{attribute 'pack_mode' := '1'} 
// ------------------------------------------------------------------------- 
//  SRCI Robot Library                                                
// ------------------------------------------------------------------------- 
//                                                                           
//  Object:      ReadAnalogInputOutCmd                                       
//  Author:      Thorsten Brach                                                
//  Date:        2024-08-09
//
//  Description:                                              
//   
//                                                                           
//  Copyright: 
//    (C) 2024 Thorsten Brach. All rights reserved                                                                                                                                            
//             Licensed under the MIT License.
//                                                                           
//  Disclaimer:                                                                           
//    This project is provided without any guarantee and can be used for   
//    private and commercial purposes. Any use is at the user’s 
//    own risk and responsibility.
//
// -------------------------------------------------------------------------
TYPE ReadAnalogInputOutCmd :
STRUCT
  /// Relates to ListenerID >0 
  /// Number of successful trigger -based command invocations
  /// For more information refer to chapter 5.5.12.4.
  InvocationCounter  : USINT;
  /// Unique system-generated ID of the "Action" when the function is triggered.
  /// • >0: The "Action" is started by the trigger funcrion with identical FollowID.
  /// • <0: The "Action" is stopped by the trigger function with identical FollowID.
  /// For more information see chapter 5.5.12.4 EmitterID, ListenerID, FollowID and OriginID
  OriginID           : INT;
  /// Returned values of digital inputs
  /// Returned values of digital inputs
  /// Unit of returned Value
  Unit               : UnitType;
  /// Returned value of analog input
  Value              : REAL;
END_STRUCT
END_TYPE

{attribute 'pack_mode' := '1'} 
// ------------------------------------------------------------------------- 
//  SRCI Robot Library                                                
// ------------------------------------------------------------------------- 
//                                                                           
//  Object:      ReadAnalogInputParCmd                                       
//  Author:      Thorsten Brach                                                
//  Date:        2024-08-09
//
//  Description:                                              
//   
//                                                                           
//  Copyright: 
//    (C) 2024 Thorsten Brach. All rights reserved                                                                                                                                            
//             Licensed under the MIT License.
//                                                                           
//  Disclaimer:                                                                           
//    This project is provided without any guarantee and can be used for   
//    private and commercial purposes. Any use is at the user’s 
//    own risk and responsibility.
//
// -------------------------------------------------------------------------
TYPE ReadAnalogInputParCmd :
STRUCT
  /// Number of the analog input 1..32
  Index              : USINT; 
  /// ID of associated trigger function:
  /// •  0: No Trigger (default)  No trigger related behavior
  /// • >0: Trigger - Start executing when the trigger function with the identical EmitterID is triggered.
  /// Always positive.
  /// For more information, see chapter 5.5.12 Triggers
  ListenerID         : SINT;
END_STRUCT
END_TYPE

{attribute 'pack_mode' := '1'} 
// ------------------------------------------------------------------------- 
//  SRCI Robot Library                                                
// ------------------------------------------------------------------------- 
//                                                                           
//  Object:      ReadAnalogInputRecvData                                       
//  Author:      Thorsten Brach                                                
//  Date:        2024-08-09
//
//  Description:                                              
//   
//                                                                           
//  Copyright: 
//    (C) 2024 Thorsten Brach. All rights reserved                                                                                                                                            
//             Licensed under the MIT License.
//                                                                           
//  Disclaimer:                                                                           
//    This project is provided without any guarantee and can be used for   
//    private and commercial purposes. Any use is at the user’s 
//    own risk and responsibility.
//
// -------------------------------------------------------------------------
TYPE ReadAnalogInputRecvData EXTENDS RspHeader :
STRUCT
  /// Relates to ListenerID >0
  /// Number of successful trigger-based command invocations - For more information refer TO chapter 5.5.12.4
  InvocationCounter : USINT;  
  /// Reserve
  Reserve           : SINT;
  /// Unique system-generated ID of the "Action" when the function is triggered.
  /// • >0: The "Action" is started by the trigger funcrion with identical FollowID.
  /// • <0: The "Action" is stopped by the trigger function with identical FollowID.
  /// For more information see chapter 5.5.12.4 EmitterID, ListenerID, FollowID and OriginID
  OriginID          : INT;
  /// Returned values of digital inputs
  /// Returned values of digital inputs
  /// Unit of returned Value
  Unit               : USINT;
  /// Returned value of analog input
  Value              : REAL;  
END_STRUCT
END_TYPE

{attribute 'pack_mode' := '1'}
// ------------------------------------------------------------------------- 
//  SRCI Robot Library                                                
// ------------------------------------------------------------------------- 
//                                                                           
//  Object:      ReadAnalogInputSendData                                       
//  Author:      Thorsten Brach                                                
//  Date:        2024-08-09
//
//  Description:                                              
//   
//                                                                           
//  Copyright: 
//    (C) 2024 Thorsten Brach. All rights reserved                                                                                                                                            
//             Licensed under the MIT License.
//                                                                           
//  Disclaimer:                                                                           
//    This project is provided without any guarantee and can be used for   
//    private and commercial purposes. Any use is at the user’s 
//    own risk and responsibility.
//
// -------------------------------------------------------------------------
TYPE ReadAnalogInputSendData EXTENDS CmdHeader: 
STRUCT
  /// ID of Action that will be executed when this command is active
  /// • >0: Start Action - Start executing the Action function with the identical ListenerID.
  /// • <0: Stop Action  -  Stop executing the Action function with the identical ListenerID.
  /// • 0: No trigger (default)-  If no EmitterID is defined, the function will not trigger any Action during its execution
  /// For more information see section Triggers of this chapter or chapter 5.5.12.4.
  EmitterID          : ARRAY [0..3] OF SINT;
  /// ID of associated trigger function:
  /// •  0: No Trigger (default)  No trigger related behavior
  /// • >0: Trigger - Start executing when the trigger function with the identical EmitterID is triggered.
  /// Always positive.
  /// For more information, see chapter 5.5.12 Triggers
  ListenerID         : SINT;
  /// Reserve
  Reserve            : BYTE;
  /// Number of the analog input 1..32
  Index              : USINT; 
END_STRUCT
END_TYPE

{attribute 'pack_mode' := '1'} 
// ------------------------------------------------------------------------- 
//  SRCI Robot Library                                                
// ------------------------------------------------------------------------- 
//                                                                           
//  Object:      ReadDigitalInputsOutCmd                                       
//  Author:      Thorsten Brach                                                
//  Date:        2024-08-09
//
//  Description:                                              
//   
//                                                                           
//  Copyright: 
//    (C) 2024 Thorsten Brach. All rights reserved                                                                                                                                            
//             Licensed under the MIT License.
//                                                                           
//  Disclaimer:                                                                           
//    This project is provided without any guarantee and can be used for   
//    private and commercial purposes. Any use is at the user’s 
//    own risk and responsibility.
//
// -------------------------------------------------------------------------
TYPE ReadDHParameterOutCmd :
STRUCT
  /// Denavit–Hartenberg parameter
  DHParameter : DHParameter;
END_STRUCT
END_TYPE

{attribute 'pack_mode' := '1'} 
// ------------------------------------------------------------------------- 
//  SRCI Robot Library                                                
// ------------------------------------------------------------------------- 
//                                                                           
//  Object:      ReadDigitalInputsParCmd                                       
//  Author:      Thorsten Brach                                                
//  Date:        2024-08-09
//
//  Description:                                              
//   
//                                                                           
//  Copyright: 
//    (C) 2024 Thorsten Brach. All rights reserved                                                                                                                                            
//             Licensed under the MIT License.
//                                                                           
//  Disclaimer:                                                                           
//    This project is provided without any guarantee and can be used for   
//    private and commercial purposes. Any use is at the user’s 
//    own risk and responsibility.
//
// -------------------------------------------------------------------------
TYPE ReadDHParameterParCmd :
STRUCT
  /// Determines if returned DH parameters use modified convention or classic convention.
  /// • 0: Classic convention (default)
  /// • 1: Modified convention
  ModifiedConvention : BOOL;  
END_STRUCT
END_TYPE

{attribute 'pack_mode' := '1'} 
// ------------------------------------------------------------------------- 
//  SRCI Robot Library                                                
// ------------------------------------------------------------------------- 
//                                                                           
//  Object:      ReadDigitalInputsRecvData                                       
//  Author:      Thorsten Brach                                                
//  Date:        2024-08-09
//
//  Description:                                              
//   
//                                                                           
//  Copyright: 
//    (C) 2024 Thorsten Brach. All rights reserved                                                                                                                                            
//             Licensed under the MIT License.
//                                                                           
//  Disclaimer:                                                                           
//    This project is provided without any guarantee and can be used for   
//    private and commercial purposes. Any use is at the user’s 
//    own risk and responsibility.
//
// -------------------------------------------------------------------------
TYPE ReadDHParameterRecvData EXTENDS RspHeader :
STRUCT
  /// Denavit–Hartenberg parameter
  DHParameter : DHParameter;  
END_STRUCT
END_TYPE

{attribute 'pack_mode' := '1'}
// ------------------------------------------------------------------------- 
//  SRCI Robot Library                                                
// ------------------------------------------------------------------------- 
//                                                                           
//  Object:      ReadDigitalInputsSendData                                       
//  Author:      Thorsten Brach                                                
//  Date:        2024-08-09
//
//  Description:                                              
//   
//                                                                           
//  Copyright: 
//    (C) 2024 Thorsten Brach. All rights reserved                                                                                                                                            
//             Licensed under the MIT License.
//                                                                           
//  Disclaimer:                                                                           
//    This project is provided without any guarantee and can be used for   
//    private and commercial purposes. Any use is at the user’s 
//    own risk and responsibility.
//
// -------------------------------------------------------------------------
TYPE ReadDHParameterSendData EXTENDS CmdHeader: 
STRUCT
  /// Determines if returned DH parameters use modified convention or classic convention.
  /// • 0: Classic convention (default)
  /// • 1: Modified convention
  ModifiedConvention : BOOL;  
END_STRUCT
END_TYPE

{attribute 'pack_mode' := '1'} 
// ------------------------------------------------------------------------- 
//  SRCI Robot Library                                                
// ------------------------------------------------------------------------- 
//                                                                           
//  Object:      ReadDigitalInputsOutCmd                                       
//  Author:      Thorsten Brach                                                
//  Date:        2024-08-09
//
//  Description:                                              
//   
//                                                                           
//  Copyright: 
//    (C) 2024 Thorsten Brach. All rights reserved                                                                                                                                            
//             Licensed under the MIT License.
//                                                                           
//  Disclaimer:                                                                           
//    This project is provided without any guarantee and can be used for   
//    private and commercial purposes. Any use is at the user’s 
//    own risk and responsibility.
//
// -------------------------------------------------------------------------
TYPE ReadDigitalInputsOutCmd :
STRUCT
  /// Relates to ListenerID >0 
  /// Number of successful trigger -based command invocations
  /// For more information refer to chapter 5.5.12.4.
  InvocationCounter  : USINT;
  /// Unique system-generated ID of the "Action" when the function is triggered.
  /// • >0: The "Action" is started by the trigger funcrion with identical FollowID.
  /// • <0: The "Action" is stopped by the trigger function with identical FollowID.
  /// For more information see chapter 5.5.12.4 EmitterID, ListenerID, FollowID and OriginID
  OriginID           : INT;
  /// Returned values of digital inputs
  Values             : ARRAY[0..4] OF BYTE;
  /// Unique system-generated ID of the "Action" when the function is triggered.
  /// • >0: The "Action" is started by the trigger function with identical FollowID.
  /// • <0: The "Action" is stopped by the trigger function with identical FollowID.
  /// For more information see chapter 5.5.12.4.
END_STRUCT
END_TYPE

{attribute 'pack_mode' := '1'} 
// ------------------------------------------------------------------------- 
//  SRCI Robot Library                                                
// ------------------------------------------------------------------------- 
//                                                                           
//  Object:      ReadDigitalInputsParCmd                                       
//  Author:      Thorsten Brach                                                
//  Date:        2024-08-09
//
//  Description:                                              
//   
//                                                                           
//  Copyright: 
//    (C) 2024 Thorsten Brach. All rights reserved                                                                                                                                            
//             Licensed under the MIT License.
//                                                                           
//  Disclaimer:                                                                           
//    This project is provided without any guarantee and can be used for   
//    private and commercial purposes. Any use is at the user’s 
//    own risk and responsibility.
//
// -------------------------------------------------------------------------
TYPE ReadDigitalInputsParCmd :
STRUCT
  /// Specifies the desired byte addresses that shall be read
  Index              : ARRAY[0..4] OF USINT; 
  /// ID of associated trigger function:
  /// •  0: No Trigger (default)  No trigger related behavior
  /// • >0: Trigger - Start executing when the trigger function with the identical EmitterID is triggered.
  /// Always positive.
  /// For more information, see chapter 5.5.12 Triggers
  ListenerID         : SINT;
END_STRUCT
END_TYPE

{attribute 'pack_mode' := '1'} 
// ------------------------------------------------------------------------- 
//  SRCI Robot Library                                                
// ------------------------------------------------------------------------- 
//                                                                           
//  Object:      ReadDigitalInputsRecvData                                       
//  Author:      Thorsten Brach                                                
//  Date:        2024-08-09
//
//  Description:                                              
//   
//                                                                           
//  Copyright: 
//    (C) 2024 Thorsten Brach. All rights reserved                                                                                                                                            
//             Licensed under the MIT License.
//                                                                           
//  Disclaimer:                                                                           
//    This project is provided without any guarantee and can be used for   
//    private and commercial purposes. Any use is at the user’s 
//    own risk and responsibility.
//
// -------------------------------------------------------------------------
TYPE ReadDigitalInputsRecvData EXTENDS RspHeader :
STRUCT
  /// Relates to ListenerID >0
  /// Number of successful trigger-based command invocations - For more information refer TO chapter 5.5.12.4
  InvocationCounter : USINT;  
  /// Reserve
  Reserve           : SINT;
  /// Unique system-generated ID of the "Action" when the function is triggered.
  /// • >0: The "Action" is started by the trigger funcrion with identical FollowID.
  /// • <0: The "Action" is stopped by the trigger function with identical FollowID.
  /// For more information see chapter 5.5.12.4 EmitterID, ListenerID, FollowID and OriginID
  OriginID          : INT;
  /// Returned values of digital inputs
  Values             : ARRAY[0..4] OF BYTE;
  
END_STRUCT
END_TYPE

{attribute 'pack_mode' := '1'}
// ------------------------------------------------------------------------- 
//  SRCI Robot Library                                                
// ------------------------------------------------------------------------- 
//                                                                           
//  Object:      ReadDigitalInputsSendData                                       
//  Author:      Thorsten Brach                                                
//  Date:        2024-08-09
//
//  Description:                                              
//   
//                                                                           
//  Copyright: 
//    (C) 2024 Thorsten Brach. All rights reserved                                                                                                                                            
//             Licensed under the MIT License.
//                                                                           
//  Disclaimer:                                                                           
//    This project is provided without any guarantee and can be used for   
//    private and commercial purposes. Any use is at the user’s 
//    own risk and responsibility.
//
// -------------------------------------------------------------------------
TYPE ReadDigitalInputsSendData EXTENDS CmdHeader: 
STRUCT
  /// ID of Action that will be executed when this command is active
  /// • >0: Start Action - Start executing the Action function with the identical ListenerID.
  /// • <0: Stop Action  -  Stop executing the Action function with the identical ListenerID.
  /// • 0: No trigger (default)-  If no EmitterID is defined, the function will not trigger any Action during its execution
  /// For more information see section Triggers of this chapter or chapter 5.5.12.4.
  EmitterID          : ARRAY [0..3] OF SINT;
  /// ID of associated trigger function:
  /// •  0: No Trigger (default)  No trigger related behavior
  /// • >0: Trigger - Start executing when the trigger function with the identical EmitterID is triggered.
  /// Always positive.
  /// For more information, see chapter 5.5.12 Triggers
  ListenerID         : SINT;
  /// Reserve
  Reserve            : BYTE;
  /// Specifies the desired byte addresses that shall be read
  Index              : ARRAY[0..4] OF USINT;
END_STRUCT
END_TYPE

{attribute 'pack_mode' := '1'} 
// ------------------------------------------------------------------------- 
//  SRCI Robot Library                                                
// ------------------------------------------------------------------------- 
//                                                                           
//  Object:      ReadDigitalOutputsOutCmd                                       
//  Author:      Thorsten Brach                                                
//  Date:        2024-08-09
//
//  Description:                                              
//   
//                                                                           
//  Copyright: 
//    (C) 2024 Thorsten Brach. All rights reserved                                                                                                                                            
//             Licensed under the MIT License.
//                                                                           
//  Disclaimer:                                                                           
//    This project is provided without any guarantee and can be used for   
//    private and commercial purposes. Any use is at the user’s 
//    own risk and responsibility.
//
// -------------------------------------------------------------------------
TYPE ReadDigitalOutputsOutCmd :
STRUCT
  /// Relates to ListenerID >0 
  /// Number of successful trigger -based command invocations
  /// For more information refer to chapter 5.5.12.4.
  InvocationCounter  : USINT;
  /// Unique system-generated ID of the "Action" when the function is triggered.
  /// • >0: The "Action" is started by the trigger funcrion with identical FollowID.
  /// • <0: The "Action" is stopped by the trigger function with identical FollowID.
  /// For more information see chapter 5.5.12.4 EmitterID, ListenerID, FollowID and OriginID
  OriginID           : INT;
  /// Returned values of digital inputs
  Values             : ARRAY[0..4] OF BYTE;
END_STRUCT
END_TYPE

{attribute 'pack_mode' := '1'} 
// ------------------------------------------------------------------------- 
//  SRCI Robot Library                                                
// ------------------------------------------------------------------------- 
//                                                                           
//  Object:      ReadDigitalOutputsParCmd                                       
//  Author:      Thorsten Brach                                                
//  Date:        2024-08-09
//
//  Description:                                              
//   
//                                                                           
//  Copyright: 
//    (C) 2024 Thorsten Brach. All rights reserved                                                                                                                                            
//             Licensed under the MIT License.
//                                                                           
//  Disclaimer:                                                                           
//    This project is provided without any guarantee and can be used for   
//    private and commercial purposes. Any use is at the user’s 
//    own risk and responsibility.
//
// -------------------------------------------------------------------------
TYPE ReadDigitalOutputsParCmd :
STRUCT
  /// Specifies the desired byte addresses that shall be read
  Index              : ARRAY[0..4] OF USINT; 
  /// ID of associated trigger function:
  /// •  0: No Trigger (default)  No trigger related behavior
  /// • >0: Trigger - Start executing when the trigger function with the identical EmitterID is triggered.
  /// Always positive.
  /// For more information, see chapter 5.5.12 Triggers
  ListenerID         : SINT;
END_STRUCT
END_TYPE

{attribute 'pack_mode' := '1'} 
// ------------------------------------------------------------------------- 
//  SRCI Robot Library                                                
// ------------------------------------------------------------------------- 
//                                                                           
//  Object:      ReadDigitalOutputsRecvData                                       
//  Author:      Thorsten Brach                                                
//  Date:        2024-08-09
//
//  Description:                                              
//   
//                                                                           
//  Copyright: 
//    (C) 2024 Thorsten Brach. All rights reserved                                                                                                                                            
//             Licensed under the MIT License.
//                                                                           
//  Disclaimer:                                                                           
//    This project is provided without any guarantee and can be used for   
//    private and commercial purposes. Any use is at the user’s 
//    own risk and responsibility.
//
// -------------------------------------------------------------------------
TYPE ReadDigitalOutputsRecvData EXTENDS RspHeader :
STRUCT
  /// Relates to ListenerID >0
  /// Number of successful trigger-based command invocations - For more information refer TO chapter 5.5.12.4
  InvocationCounter : USINT;  
  /// Reserve
  Reserve           : SINT;
  /// Unique system-generated ID of the "Action" when the function is triggered.
  /// • >0: The "Action" is started by the trigger funcrion with identical FollowID.
  /// • <0: The "Action" is stopped by the trigger function with identical FollowID.
  /// For more information see chapter 5.5.12.4 EmitterID, ListenerID, FollowID and OriginID
  OriginID          : INT;
  /// Returned values of digital inputs
  Values             : ARRAY[0..4] OF BYTE;
END_STRUCT
END_TYPE

{attribute 'pack_mode' := '1'}
// ------------------------------------------------------------------------- 
//  SRCI Robot Library                                                
// ------------------------------------------------------------------------- 
//                                                                           
//  Object:      ReadDigitalOutputsSendData                                       
//  Author:      Thorsten Brach                                                
//  Date:        2024-08-09
//
//  Description:                                              
//   
//                                                                           
//  Copyright: 
//    (C) 2024 Thorsten Brach. All rights reserved                                                                                                                                            
//             Licensed under the MIT License.
//                                                                           
//  Disclaimer:                                                                           
//    This project is provided without any guarantee and can be used for   
//    private and commercial purposes. Any use is at the user’s 
//    own risk and responsibility.
//
// -------------------------------------------------------------------------
TYPE ReadDigitalOutputsSendData EXTENDS CmdHeader: 
STRUCT
  /// ID of Action that will be executed when this command is active
  /// • >0: Start Action - Start executing the Action function with the identical ListenerID.
  /// • <0: Stop Action  -  Stop executing the Action function with the identical ListenerID.
  /// • 0: No trigger (default)-  If no EmitterID is defined, the function will not trigger any Action during its execution
  /// For more information see section Triggers of this chapter or chapter 5.5.12.4.
  EmitterID          : ARRAY [0..3] OF SINT;
  /// ID of associated trigger function:
  /// •  0: No Trigger (default)  No trigger related behavior
  /// • >0: Trigger - Start executing when the trigger function with the identical EmitterID is triggered.
  /// Always positive.
  /// For more information, see chapter 5.5.12 Triggers
  ListenerID         : SINT;
  /// Reserve
  Reserve            : BYTE;
  /// Specifies the desired byte addresses that shall be read
  Index              : ARRAY[0..4] OF USINT; 
END_STRUCT
END_TYPE

{attribute 'pack_mode' := '1'} 
// ------------------------------------------------------------------------- 
//  SRCI Robot Library                                                
// ------------------------------------------------------------------------- 
//                                                                           
//  Object:      ReadDigitalOutputsOutCmd                                       
//  Author:      Thorsten Brach                                                
//  Date:        2024-08-09
//
//  Description:                                              
//   
//                                                                           
//  Copyright: 
//    (C) 2024 Thorsten Brach. All rights reserved                                                                                                                                            
//             Licensed under the MIT License.
//                                                                           
//  Disclaimer:                                                                           
//    This project is provided without any guarantee and can be used for   
//    private and commercial purposes. Any use is at the user’s 
//    own risk and responsibility.
//
// -------------------------------------------------------------------------
TYPE ReadFrameDataOutCmd :
STRUCT
  /// Frame index
  FrameNoReturn      : USINT;
  /// Frame data (see chapter 5.5.6.2)
  FrameData          : FrameData;
END_STRUCT
END_TYPE

{attribute 'pack_mode' := '1'} 
// ------------------------------------------------------------------------- 
//  SRCI Robot Library                                                
// ------------------------------------------------------------------------- 
//                                                                           
//  Object:      ReadDigitalOutputsParCmd                                       
//  Author:      Thorsten Brach                                                
//  Date:        2024-08-09
//
//  Description:                                              
//   
//                                                                           
//  Copyright: 
//    (C) 2024 Thorsten Brach. All rights reserved                                                                                                                                            
//             Licensed under the MIT License.
//                                                                           
//  Disclaimer:                                                                           
//    This project is provided without any guarantee and can be used for   
//    private and commercial purposes. Any use is at the user’s 
//    own risk and responsibility.
//
// -------------------------------------------------------------------------
TYPE ReadFrameDataParCmd :
STRUCT
  /// Frame index
  /// • -1: Currently used frame on RC
  /// • 0: WCS
  /// • 1 (default)..254: UCS (User frames)
  FrameNo            : INT;
END_STRUCT
END_TYPE

{attribute 'pack_mode' := '1'} 
// ------------------------------------------------------------------------- 
//  SRCI Robot Library                                                
// ------------------------------------------------------------------------- 
//                                                                           
//  Object:      ReadDigitalOutputsRecvData                                       
//  Author:      Thorsten Brach                                                
//  Date:        2024-08-09
//
//  Description:                                              
//   
//                                                                           
//  Copyright: 
//    (C) 2024 Thorsten Brach. All rights reserved                                                                                                                                            
//             Licensed under the MIT License.
//                                                                           
//  Disclaimer:                                                                           
//    This project is provided without any guarantee and can be used for   
//    private and commercial purposes. Any use is at the user’s 
//    own risk and responsibility.
//
// -------------------------------------------------------------------------
TYPE ReadFrameDataRecvData EXTENDS RspHeader :
STRUCT
  /// Reserve
  Reserve       : BYTE;
  /// Frame index
  FrameNoReturn : USINT;
  /// Frame data (see chapter 5.5.6.2)
  FrameData     : FrameData;
  /// The status bit "DataChanged" represents the modification state 
  DataChanged   : BOOL;
END_STRUCT
END_TYPE

{attribute 'pack_mode' := '1'}
// ------------------------------------------------------------------------- 
//  SRCI Robot Library                                                
// ------------------------------------------------------------------------- 
//                                                                           
//  Object:      ReadDigitalOutputsSendData                                       
//  Author:      Thorsten Brach                                                
//  Date:        2024-08-09
//
//  Description:                                              
//   
//                                                                           
//  Copyright: 
//    (C) 2024 Thorsten Brach. All rights reserved                                                                                                                                            
//             Licensed under the MIT License.
//                                                                           
//  Disclaimer:                                                                           
//    This project is provided without any guarantee and can be used for   
//    private and commercial purposes. Any use is at the user’s 
//    own risk and responsibility.
//
// -------------------------------------------------------------------------
TYPE ReadFrameDataSendData EXTENDS CmdHeader: 
STRUCT
  /// Frame index
  /// • -1: Currently used frame on RC
  /// • 0: WCS
  /// • 1 (default)..254: UCS (User frames)
  FrameNo            : USINT;
END_STRUCT
END_TYPE

{attribute 'pack_mode' := '1'} 
// ------------------------------------------------------------------------- 
//  SRCI Robot Library                                                
// ------------------------------------------------------------------------- 
//                                                                           
//  Object:      ReadIntegersOutCmd                                       
//  Author:      Thorsten Brach                                                
//  Date:        2024-08-09
//
//  Description:                                              
//   
//                                                                           
//  Copyright: 
//    (C) 2024 Thorsten Brach. All rights reserved                                                                                                                                            
//             Licensed under the MIT License.
//                                                                           
//  Disclaimer:                                                                           
//    This project is provided without any guarantee and can be used for   
//    private and commercial purposes. Any use is at the user’s 
//    own risk and responsibility.
//
// -------------------------------------------------------------------------
TYPE ReadIntegersOutCmd :
STRUCT
  /// Returned values of integer register
  Values             : ARRAY[0..6] OF INT;
  /// Unique system-generated ID of the "Action" when the function is triggered.
  /// • >0: The "Action" is started by the trigger function with identical FollowID.
  /// • <0: The "Action" is stopped by the trigger function with identical FollowID.
  /// For more information see chapter 5.5.12.4.
  OriginID           : INT;
  /// Relates to ListenerID >0 
  /// Number of successful trigger -based command invocations
  /// For more information refer to chapter 5.5.12.4.
  InvocationCounter  : USINT;
END_STRUCT
END_TYPE

{attribute 'pack_mode' := '1'} 
// ------------------------------------------------------------------------- 
//  SRCI Robot Library                                                
// ------------------------------------------------------------------------- 
//                                                                           
//  Object:      ReadIntegersParCmd                                       
//  Author:      Thorsten Brach                                                
//  Date:        2024-08-09
//
//  Description:                                              
//   
//                                                                           
//  Copyright: 
//    (C) 2024 Thorsten Brach. All rights reserved                                                                                                                                            
//             Licensed under the MIT License.
//                                                                           
//  Disclaimer:                                                                           
//    This project is provided without any guarantee and can be used for   
//    private and commercial purposes. Any use is at the user’s 
//    own risk and responsibility.
//
// -------------------------------------------------------------------------
TYPE ReadIntegersParCmd :
STRUCT
  /// Specifies the desired target values that shall be read
  Index              : ARRAY[0..6] OF USINT; 
  /// ID of associated trigger function:
  /// •  0: No Trigger (default)  No trigger related behavior
  /// • >0: Trigger - Start executing when the trigger function with the identical EmitterID is triggered.
  /// Always positive.
  /// For more information, see chapter 5.5.12 Triggers
  ListenerID         : SINT;
END_STRUCT
END_TYPE

{attribute 'pack_mode' := '1'} 
// ------------------------------------------------------------------------- 
//  SRCI Robot Library                                                
// ------------------------------------------------------------------------- 
//                                                                           
//  Object:      ReadIntegersRecvData                                       
//  Author:      Thorsten Brach                                                
//  Date:        2024-08-09
//
//  Description:                                              
//   
//                                                                           
//  Copyright: 
//    (C) 2024 Thorsten Brach. All rights reserved                                                                                                                                            
//             Licensed under the MIT License.
//                                                                           
//  Disclaimer:                                                                           
//    This project is provided without any guarantee and can be used for   
//    private and commercial purposes. Any use is at the user’s 
//    own risk and responsibility.
//
// -------------------------------------------------------------------------
TYPE ReadIntegersRecvData EXTENDS RspHeader :
STRUCT
  /// Relates to ListenerID >0 
  /// Number of successful trigger -based command invocations
  /// For more information refer to chapter 5.5.12.4.
  InvocationCounter  : USINT;
  /// Reserve
  Reserve            : BYTE;
  /// Unique system-generated ID of the "Action" when the function is triggered.
  /// • >0: The "Action" is started by the trigger function with identical FollowID.
  /// • <0: The "Action" is stopped by the trigger function with identical FollowID.
  /// For more information see chapter 5.5.12.4.
  OriginID           : INT;
  /// Returned values of integer register
  Values             : ARRAY[0..6] OF INT;
END_STRUCT
END_TYPE

{attribute 'pack_mode' := '1'}
// ------------------------------------------------------------------------- 
//  SRCI Robot Library                                                
// ------------------------------------------------------------------------- 
//                                                                           
//  Object:      ReadIntegersSendData                                       
//  Author:      Thorsten Brach                                                
//  Date:        2024-08-09
//
//  Description:                                              
//   
//                                                                           
//  Copyright: 
//    (C) 2024 Thorsten Brach. All rights reserved                                                                                                                                            
//             Licensed under the MIT License.
//                                                                           
//  Disclaimer:                                                                           
//    This project is provided without any guarantee and can be used for   
//    private and commercial purposes. Any use is at the user’s 
//    own risk and responsibility.
//
// -------------------------------------------------------------------------
TYPE ReadIntegersSendData EXTENDS CmdHeader: 
STRUCT
  /// ID of Action that will be executed when this command is active
  /// • >0: Start Action - Start executing the Action function with the identical ListenerID.
  /// • <0: Stop Action  -  Stop executing the Action function with the identical ListenerID.
  /// • 0: No trigger (default)-  If no EmitterID is defined, the function will not trigger any Action during its execution
  /// For more information see section Triggers of this chapter or chapter 5.5.12.4.
  EmitterID          : ARRAY [0..3] OF SINT;
  /// ID of associated trigger function:
  /// •  0: No Trigger (default)  No trigger related behavior
  /// • >0: Trigger - Start executing when the trigger function with the identical EmitterID is triggered.
  /// Always positive.
  /// For more information, see chapter 5.5.12 Triggers
  ListenerID         : SINT;
  /// Reserve
  Reserve            : BYTE;  
  /// Specifies the desired target values that shall be read
  Index              : ARRAY[0..6] OF USINT; 
END_STRUCT
END_TYPE

{attribute 'pack_mode' := '1'} 
// ------------------------------------------------------------------------- 
//  SRCI Robot Library                                                
// ------------------------------------------------------------------------- 
//                                                                           
//  Object:      ReadLoadDataOutCmd                                       
//  Author:      Thorsten Brach                                                
//  Date:        2024-08-09
//
//  Description:                                              
//   
//                                                                           
//  Copyright: 
//    (C) 2024 Thorsten Brach. All rights reserved                                                                                                                                            
//             Licensed under the MIT License.
//                                                                           
//  Disclaimer:                                                                           
//    This project is provided without any guarantee and can be used for   
//    private and commercial purposes. Any use is at the user’s 
//    own risk and responsibility.
//
// -------------------------------------------------------------------------
TYPE ReadLoadDataOutCmd :
STRUCT
  /// Tool index
  LoadNoReturn       : USINT;
  /// Load data (see chapter 5.5.6.4)
  LoadData           : LoadData;
END_STRUCT
END_TYPE

{attribute 'pack_mode' := '1'} 
// ------------------------------------------------------------------------- 
//  SRCI Robot Library                                                
// ------------------------------------------------------------------------- 
//                                                                           
//  Object:      ReadLoadDataParCmd                                       
//  Author:      Thorsten Brach                                                
//  Date:        2024-08-09
//
//  Description:                                              
//   
//                                                                           
//  Copyright: 
//    (C) 2024 Thorsten Brach. All rights reserved                                                                                                                                            
//             Licensed under the MIT License.
//                                                                           
//  Disclaimer:                                                                           
//    This project is provided without any guarantee and can be used for   
//    private and commercial purposes. Any use is at the user’s 
//    own risk and responsibility.
//
// -------------------------------------------------------------------------
TYPE ReadLoadDataParCmd :
STRUCT
  /// Load index
  /// • -1: Currently used load on RC
  /// •  0: Not possible to read
  /// •  1 (default)..254: Load data
  LoadNo             : INT;
END_STRUCT
END_TYPE

{attribute 'pack_mode' := '1'} 
// ------------------------------------------------------------------------- 
//  SRCI Robot Library                                                
// ------------------------------------------------------------------------- 
//                                                                           
//  Object:      ReadLoadDataRecvData                                       
//  Author:      Thorsten Brach                                                
//  Date:        2024-08-09
//
//  Description:                                              
//   
//                                                                           
//  Copyright: 
//    (C) 2024 Thorsten Brach. All rights reserved                                                                                                                                            
//             Licensed under the MIT License.
//                                                                           
//  Disclaimer:                                                                           
//    This project is provided without any guarantee and can be used for   
//    private and commercial purposes. Any use is at the user’s 
//    own risk and responsibility.
//
// -------------------------------------------------------------------------
TYPE ReadLoadDataRecvData EXTENDS RspHeader :
STRUCT
  /// Tool index
  LoadNoReturn : USINT;
  /// Load data (see chapter 5.5.6.4)
  LoadData     : LoadData;
  /// The status bit "DataChanged" represents the modification state 
  DataChanged  : BOOL;
END_STRUCT
END_TYPE

{attribute 'pack_mode' := '1'}
// ------------------------------------------------------------------------- 
//  SRCI Robot Library                                                
// ------------------------------------------------------------------------- 
//                                                                           
//  Object:      ReadLoadDataSendData                                       
//  Author:      Thorsten Brach                                                
//  Date:        2024-08-09
//
//  Description:                                              
//   
//                                                                           
//  Copyright: 
//    (C) 2024 Thorsten Brach. All rights reserved                                                                                                                                            
//             Licensed under the MIT License.
//                                                                           
//  Disclaimer:                                                                           
//    This project is provided without any guarantee and can be used for   
//    private and commercial purposes. Any use is at the user’s 
//    own risk and responsibility.
//
// -------------------------------------------------------------------------
TYPE ReadLoadDataSendData EXTENDS CmdHeader: 
STRUCT
  /// Load index
  /// • -1: Currently used load on RC
  /// •  0: Not possible to read
  /// •  1 (default)..254: Load data
  LoadNo             : USINT;
END_STRUCT
END_TYPE

{attribute 'pack_mode' := '1'} 
// ------------------------------------------------------------------------- 
//  SRCI Robot Library                                                
// ------------------------------------------------------------------------- 
//                                                                           
//  Object:      ReadMessagesOutCmd                                       
//  Author:      Thorsten Brach                                                
//  Date:        2024-08-09
//
//  Description:                                              
//   
//                                                                           
//  Copyright: 
//    (C) 2024 Thorsten Brach. All rights reserved                                                                                                                                            
//             Licensed under the MIT License.
//                                                                           
//  Disclaimer:                                                                           
//    This project is provided without any guarantee and can be used for   
//    private and commercial purposes. Any use is at the user’s 
//    own risk and responsibility.
//
// -------------------------------------------------------------------------
TYPE ReadMessagesOutCmd :
STRUCT
  /// ID for function specific acknowledgement mechanism
  MsgId                  : USINT;
  /// Number of pending errors on RC
  NumberOfActiveErrors   : USINT;
  /// Number if pending warnings in RC
  NumberOfActiveWarnings : USINT;
  /// Timestamp
  Timestamp              : IEC_TIMESTAMP;
  /// Message Type
  MsgType                : MessageType;
  /// Severity of returned message according to .Table 5-47.
  Severity               : Severity;
  /// ErrorCode
  ErrorCode              : DWORD;
  /// Test
  Text                   : STRING(255);
END_STRUCT
END_TYPE

{attribute 'pack_mode' := '1'} 
// ------------------------------------------------------------------------- 
//  SRCI Robot Library                                                
// ------------------------------------------------------------------------- 
//                                                                           
//  Object:      ReadMessagesParCmd                                       
//  Author:      Thorsten Brach                                                
//  Date:        2024-08-09
//
//  Description:                                              
//   
//                                                                           
//  Copyright: 
//    (C) 2024 Thorsten Brach. All rights reserved                                                                                                                                            
//             Licensed under the MIT License.
//                                                                           
//  Disclaimer:                                                                           
//    This project is provided without any guarantee and can be used for   
//    private and commercial purposes. Any use is at the user’s 
//    own risk and responsibility.
//
// -------------------------------------------------------------------------
TYPE ReadMessagesParCmd :
STRUCT
  /// ID for function specific acknowledgement mechanism
  MsgID        : USINT;
  /// Defines up to which level of severity messages will be transmitted to the PLC’s message buffer
  MessageLevel : MessageLevel;
END_STRUCT
END_TYPE

{attribute 'pack_mode' := '1'} 
// ------------------------------------------------------------------------- 
//  SRCI Robot Library                                                
// ------------------------------------------------------------------------- 
//                                                                           
//  Object:      ReadMessagesRecvData                                       
//  Author:      Thorsten Brach                                                
//  Date:        2024-08-09
//
//  Description:                                              
//   
//                                                                           
//  Copyright: 
//    (C) 2024 Thorsten Brach. All rights reserved                                                                                                                                            
//             Licensed under the MIT License.
//                                                                           
//  Disclaimer:                                                                           
//    This project is provided without any guarantee and can be used for   
//    private and commercial purposes. Any use is at the user’s 
//    own risk and responsibility.
//
// -------------------------------------------------------------------------
TYPE ReadMessagesRecvData EXTENDS RspHeader :
STRUCT
  /// Set TRUE to read messages from RC.
  Enabled                : BOOL;
  /// ID for function specific acknowledgement mechanism
  MsgId                  : USINT;
  /// Number of pending errors on RC
  NumberOfActiveErrors   : USINT;
  /// Number if pending warnings in RC
  NumberOfActiveWarnings : USINT;
  /// Timestamp
  Timestamp              : IEC_TIMESTAMP;
  /// Message Type
  MsgType                : USINT;
  /// Severity of returned message according to .Table 5-47.
  Severity               : SINT;
  /// ErrorCode
  ErrorCode              : DWORD;
  /// Test
  Text                   : STRING(255);
END_STRUCT
END_TYPE

{attribute 'pack_mode' := '1'}
// ------------------------------------------------------------------------- 
//  SRCI Robot Library                                                
// ------------------------------------------------------------------------- 
//                                                                           
//  Object:      ReadMessagesSendData                                       
//  Author:      Thorsten Brach                                                
//  Date:        2024-08-09
//
//  Description:                                              
//   
//                                                                           
//  Copyright: 
//    (C) 2024 Thorsten Brach. All rights reserved                                                                                                                                            
//             Licensed under the MIT License.
//                                                                           
//  Disclaimer:                                                                           
//    This project is provided without any guarantee and can be used for   
//    private and commercial purposes. Any use is at the user’s 
//    own risk and responsibility.
//
// -------------------------------------------------------------------------
TYPE ReadMessagesSendData EXTENDS CmdHeader: 
STRUCT
  /// ID for function specific acknowledgement mechanism
  MsgID        : USINT;
  /// TRUE when function is returning messages from RC
  Enable       : BOOL;
  /// Defines up to which level of severity messages will be transmitted to the PLC’s message buffer
  MessageLevel : USINT;
END_STRUCT
END_TYPE

{attribute 'pack_mode' := '1'} 
// ------------------------------------------------------------------------- 
//  SRCI Robot Library                                                
// ------------------------------------------------------------------------- 
//                                                                           
//  Object:      ReadRealsOutCmd                                       
//  Author:      Thorsten Brach                                                
//  Date:        2024-08-09
//
//  Description:                                              
//   
//                                                                           
//  Copyright: 
//    (C) 2024 Thorsten Brach. All rights reserved                                                                                                                                            
//             Licensed under the MIT License.
//                                                                           
//  Disclaimer:                                                                           
//    This project is provided without any guarantee and can be used for   
//    private and commercial purposes. Any use is at the user’s 
//    own risk and responsibility.
//
// -------------------------------------------------------------------------
TYPE ReadRealsOutCmd :
STRUCT
  /// Relates to ListenerID >0 
  /// Number of successful trigger -based command invocations
  /// For more information refer to chapter 5.5.12.4.
  InvocationCounter  : USINT;
  /// Unique system-generated ID of the "Action" when the function is triggered.
  /// • >0: The "Action" is started by the trigger function with identical FollowID.
  /// • <0: The "Action" is stopped by the trigger function with identical FollowID.
  /// For more information see chapter 5.5.12.4.
  OriginID           : INT;
  /// Returned values of real register
  Values             : ARRAY[0..6] OF REAL;
END_STRUCT
END_TYPE

{attribute 'pack_mode' := '1'} 
// ------------------------------------------------------------------------- 
//  SRCI Robot Library                                                
// ------------------------------------------------------------------------- 
//                                                                           
//  Object:      ReadRealsParCmd                                       
//  Author:      Thorsten Brach                                                
//  Date:        2024-08-09
//
//  Description:                                              
//   
//                                                                           
//  Copyright: 
//    (C) 2024 Thorsten Brach. All rights reserved                                                                                                                                            
//             Licensed under the MIT License.
//                                                                           
//  Disclaimer:                                                                           
//    This project is provided without any guarantee and can be used for   
//    private and commercial purposes. Any use is at the user’s 
//    own risk and responsibility.
//
// -------------------------------------------------------------------------
TYPE ReadRealsParCmd :
STRUCT
  /// Specifies the desired target values that shall be read
  Index              : ARRAY[0..6] OF USINT; 
  /// ID of associated trigger function:
  /// •  0: No Trigger (default)  No trigger related behavior
  /// • >0: Trigger - Start executing when the trigger function with the identical EmitterID is triggered.
  /// Always positive.
  /// For more information, see chapter 5.5.12 Triggers
  ListenerID         : SINT;
END_STRUCT
END_TYPE

{attribute 'pack_mode' := '1'} 
// ------------------------------------------------------------------------- 
//  SRCI Robot Library                                                
// ------------------------------------------------------------------------- 
//                                                                           
//  Object:      ReadRealsRecvData                                       
//  Author:      Thorsten Brach                                                
//  Date:        2024-08-09
//
//  Description:                                              
//   
//                                                                           
//  Copyright: 
//    (C) 2024 Thorsten Brach. All rights reserved                                                                                                                                            
//             Licensed under the MIT License.
//                                                                           
//  Disclaimer:                                                                           
//    This project is provided without any guarantee and can be used for   
//    private and commercial purposes. Any use is at the user’s 
//    own risk and responsibility.
//
// -------------------------------------------------------------------------
TYPE ReadRealsRecvData EXTENDS RspHeader :
STRUCT
  /// Relates to ListenerID >0 
  /// Number of successful trigger -based command invocations
  /// For more information refer to chapter 5.5.12.4.
  InvocationCounter  : USINT;
  /// Reserve
  Reserve            : SINT;
  /// Unique system-generated ID of the "Action" when the function is triggered.
  /// • >0: The "Action" is started by the trigger function with identical FollowID.
  /// • <0: The "Action" is stopped by the trigger function with identical FollowID.
  /// For more information see chapter 5.5.12.4.
  OriginID           : INT;
  /// Returned values of real register
  Values             : ARRAY[0..6] OF REAL;
END_STRUCT
END_TYPE

{attribute 'pack_mode' := '1'}
// ------------------------------------------------------------------------- 
//  SRCI Robot Library                                                
// ------------------------------------------------------------------------- 
//                                                                           
//  Object:      ReadRealsSendData                                       
//  Author:      Thorsten Brach                                                
//  Date:        2024-08-09
//
//  Description:                                              
//   
//                                                                           
//  Copyright: 
//    (C) 2024 Thorsten Brach. All rights reserved                                                                                                                                            
//             Licensed under the MIT License.
//                                                                           
//  Disclaimer:                                                                           
//    This project is provided without any guarantee and can be used for   
//    private and commercial purposes. Any use is at the user’s 
//    own risk and responsibility.
//
// -------------------------------------------------------------------------
TYPE ReadRealsSendData EXTENDS CmdHeader: 
STRUCT
  /// ID of Action that will be executed when this command is active
  /// • >0: Start Action - Start executing the Action function with the identical ListenerID.
  /// • <0: Stop Action  -  Stop executing the Action function with the identical ListenerID.
  /// • 0: No trigger (default)-  If no EmitterID is defined, the function will not trigger any Action during its execution
  /// For more information see section Triggers of this chapter or chapter 5.5.12.4.
  EmitterID          : ARRAY [0..3] OF SINT;  
  /// ID of associated trigger function:
  /// • 0: Immediately (default) - Start executing this function immediately.
  /// • >0: Trigger -  Start executing, when the trigger function with the identical EmitterID is triggered.
  /// Always positive.
  /// For more information, see chapter 5.5.12 Triggers
  ListenerID         : SINT;
  /// Reserve
  Reserve            : SINT;
  /// Specifies the desired target values that shall be read
  Index              : ARRAY[0..6] OF USINT; 
END_STRUCT
END_TYPE

{attribute 'pack_mode' := '1'} 
// ------------------------------------------------------------------------- 
//  SRCI Robot Library                                                
// ------------------------------------------------------------------------- 
//                                                                           
//  Object:      ReadRealsOutCmd                                       
//  Author:      Thorsten Brach                                                
//  Date:        2024-08-09
//
//  Description:                                              
//   
//                                                                           
//  Copyright: 
//    (C) 2024 Thorsten Brach. All rights reserved                                                                                                                                            
//             Licensed under the MIT License.
//                                                                           
//  Disclaimer:                                                                           
//    This project is provided without any guarantee and can be used for   
//    private and commercial purposes. Any use is at the user’s 
//    own risk and responsibility.
//
// -------------------------------------------------------------------------
TYPE ReadRobotDataOutCmd :
STRUCT
  /// RC manufacturer name
  RCManufacturer       : STRING(20);
  /// RC part number
  RCOrderID            : STRING(20);
  /// RC serial number
  RCSerialNumber       : STRING(16);
  /// RA serial number
  RASerialNumber       : STRING(16);
  /// Robot firmware version in manufacturer -specific format
  RCFirmwareVersion    : STRING(12);
  /// 
  RCInterpreterVersion : STRING(5);
  /// TRUE = Axis used in Robot FALSE = Axis NOT used. See Table 6-13 for bit assignment
  AxisJointUsed        : AxisJointUsed;
  /// TRUE = Axis used by Robot FALSE = Axis NOT used. See Table 6-13 for bit assignment.
  AxisExternalUsed     : AxisExternalUsed;
  /// TRUE = mm FALSE = ° See Table 6-13 for bit assignment.
  AxisJointUnit        : AxisJointUnit;
  /// TRUE = mm FALSE = ° See Table 6-13 for bit assignment
  AxisExternalUnit     : AxisExternalUnit;
  /// • TRUE: Function is supported by RC • FALSE: Function is not supported by RC See Table 6-14 for bit assignment.
  RCSupportedFunctions  : RCSupportedFunctions;
  /// Unique and unmodifiable identification of the RA.
  RobotID              : STRING(16);  
  /// Interpreter task cycle time of the RC [ms]
  InterpreterCycleTime : UINT;
END_STRUCT
END_TYPE

{attribute 'pack_mode' := '1'} 
// ------------------------------------------------------------------------- 
//  SRCI Robot Library                                                
// ------------------------------------------------------------------------- 
//                                                                           
//  Object:      ReadRealsParCmd                                       
//  Author:      Thorsten Brach                                                
//  Date:        2024-08-09
//
//  Description:                                              
//   
//                                                                           
//  Copyright: 
//    (C) 2024 Thorsten Brach. All rights reserved                                                                                                                                            
//             Licensed under the MIT License.
//                                                                           
//  Disclaimer:                                                                           
//    This project is provided without any guarantee and can be used for   
//    private and commercial purposes. Any use is at the user’s 
//    own risk and responsibility.
//
// -------------------------------------------------------------------------
TYPE ReadRobotDataParCmd :
STRUCT
END_STRUCT
END_TYPE

{attribute 'pack_mode' := '1'} 
// ------------------------------------------------------------------------- 
//  SRCI Robot Library                                                
// ------------------------------------------------------------------------- 
//                                                                           
//  Object:      ReadRealsRecvData                                       
//  Author:      Thorsten Brach                                                
//  Date:        2024-08-09
//
//  Description:                                              
//   
//                                                                           
//  Copyright: 
//    (C) 2024 Thorsten Brach. All rights reserved                                                                                                                                            
//             Licensed under the MIT License.
//                                                                           
//  Disclaimer:                                                                           
//    This project is provided without any guarantee and can be used for   
//    private and commercial purposes. Any use is at the user’s 
//    own risk and responsibility.
//
// -------------------------------------------------------------------------
TYPE ReadRobotDataRecvData EXTENDS RspHeader :
STRUCT
  /// RC manufacturer name
  RCManufacturer       : STRING(20);
  /// RC part number
  RCOrderID            : STRING(20);
  /// RC serial number
  RCSerialNumber       : STRING(16);
  /// RA serial number
  RASerialNumber       : STRING(16);
  /// Robot firmware version in manufacturer -specific format
  RCFirmwareVersion    : STRING(12);
  /// 
  RCInterpreterVersion : STRING(5);
  /// Reserve
  Reserve              : BYTE;
  /// TRUE = Axis used in Robot FALSE = Axis NOT used. See Table 6-13 for bit assignment
  AxisJointUsed        : BYTE;
  /// TRUE = Axis used by Robot FALSE = Axis NOT used. See Table 6-13 for bit assignment.
  AxisExternalUsed     : BYTE;
  /// TRUE = mm FALSE = ° See Table 6-13 for bit assignment.
  AxisJointUnit        : BYTE;
  /// TRUE = mm FALSE = ° See Table 6-13 for bit assignment
  AxisExternalUnit     : BYTE;
  /// • TRUE: Function is supported by RC • FALSE: Function is not supported by RC See Table 6-14 for bit assignment.
  RCSupportedFunctions : ARRAY[0..18] OF BYTE;
  /// Reserve 2 
  Reserve2             : BYTE;
  /// Unique and unmodifiable identification of the RA.
  RobotID              : STRING(16);  
  /// Interpreter task cycle time of the RC [ms]
  InterpreterCycleTime : UINT;
END_STRUCT
END_TYPE

{attribute 'pack_mode' := '1'}
// ------------------------------------------------------------------------- 
//  SRCI Robot Library                                                
// ------------------------------------------------------------------------- 
//                                                                           
//  Object:      ReadRealsSendData                                       
//  Author:      Thorsten Brach                                                
//  Date:        2024-08-09
//
//  Description:                                              
//   
//                                                                           
//  Copyright: 
//    (C) 2024 Thorsten Brach. All rights reserved                                                                                                                                            
//             Licensed under the MIT License.
//                                                                           
//  Disclaimer:                                                                           
//    This project is provided without any guarantee and can be used for   
//    private and commercial purposes. Any use is at the user’s 
//    own risk and responsibility.
//
// -------------------------------------------------------------------------
TYPE ReadRobotDataSendData EXTENDS CmdHeader: 
STRUCT
END_STRUCT
END_TYPE

{attribute 'pack_mode' := '1'} 
// ------------------------------------------------------------------------- 
//  SRCI Robot Library                                                
// ------------------------------------------------------------------------- 
//                                                                           
//  Object:      ReadRobotDefaultDynamicsOutCmd                                       
//  Author:      Thorsten Brach                                                
//  Date:        2024-08-09
//
//  Description:                                              
//   
//                                                                           
//  Copyright: 
//    (C) 2024 Thorsten Brach. All rights reserved                                                                                                                                            
//             Licensed under the MIT License.
//                                                                           
//  Disclaimer:                                                                           
//    This project is provided without any guarantee and can be used for   
//    private and commercial purposes. Any use is at the user’s 
//    own risk and responsibility.
//
// -------------------------------------------------------------------------
TYPE ReadRobotDefaultDynamicsOutCmd :
STRUCT
  /// Default dynamics values according to Table 6-148.
  DynamicValues      : DefaultDynamics;
END_STRUCT
END_TYPE

{attribute 'pack_mode' := '1'} 
// ------------------------------------------------------------------------- 
//  SRCI Robot Library                                                
// ------------------------------------------------------------------------- 
//                                                                           
//  Object:      ReadRobotDefaultDynamicsParCmd                                       
//  Author:      Thorsten Brach                                                
//  Date:        2024-08-09
//
//  Description:                                              
//   
//                                                                           
//  Copyright: 
//    (C) 2024 Thorsten Brach. All rights reserved                                                                                                                                            
//             Licensed under the MIT License.
//                                                                           
//  Disclaimer:                                                                           
//    This project is provided without any guarantee and can be used for   
//    private and commercial purposes. Any use is at the user’s 
//    own risk and responsibility.
//
// -------------------------------------------------------------------------
TYPE ReadRobotDefaultDynamicsParCmd :
STRUCT
END_STRUCT
END_TYPE

{attribute 'pack_mode' := '1'} 
// ------------------------------------------------------------------------- 
//  SRCI Robot Library                                                
// ------------------------------------------------------------------------- 
//                                                                           
//  Object:      ReadRobotDefaultDynamicsRecvData                                       
//  Author:      Thorsten Brach                                                
//  Date:        2024-08-09
//
//  Description:                                              
//   
//                                                                           
//  Copyright: 
//    (C) 2024 Thorsten Brach. All rights reserved                                                                                                                                            
//             Licensed under the MIT License.
//                                                                           
//  Disclaimer:                                                                           
//    This project is provided without any guarantee and can be used for   
//    private and commercial purposes. Any use is at the user’s 
//    own risk and responsibility.
//
// -------------------------------------------------------------------------
TYPE ReadRobotDefaultDynamicsRecvData EXTENDS RspHeader :
STRUCT
  /// Timestamp
  Timestamp        : IEC_TIMESTAMP;
  /// Maximum velocity for the axes.
  /// Range [%]: 
  /// •  <0% : Use default velocity given by the user
  /// •   0% : Use internal minimal velocity
  /// • 100% : Use the entire reference velocity, given by the user
  VelocityRate     : UINT;
  /// Maximum acceleration.
  /// Range [%]:
  /// •  <0% : Use default acceleration given by the user
  /// •   0% : Use internal minimal acceleration
  /// • 100% : Use the entire reference acceleration, given by the user
  AccelerationRate : UINT;
  /// Maximum deceleration.
  /// Range [%] : 
  /// •  <0% : Use default deceleration given by the user
  /// •   0% : Use internal minimal deceleration
  /// • 100% : Use the entire reference deceleration, given by the user
  DecelerationRate : UINT;
  /// Maximum jerk
  /// Range [%] : 
  /// •  <0% : Use default jerk given by the user
  /// •   0% : Use internal minimal jerk
  /// • 100% : Use the entire reference jerk, given by the user (Trapezoidal if possible) 
  JerkRate         : UINT;  
  /// The status bit "DataChanged" represents the modification state 
  DataChanged      : BOOL;
END_STRUCT
END_TYPE

{attribute 'pack_mode' := '1'}
// ------------------------------------------------------------------------- 
//  SRCI Robot Library                                                
// ------------------------------------------------------------------------- 
//                                                                           
//  Object:      ReadRobotDefaultDynamicsSendData                                       
//  Author:      Thorsten Brach                                                
//  Date:        2024-08-09
//
//  Description:                                              
//   
//                                                                           
//  Copyright: 
//    (C) 2024 Thorsten Brach. All rights reserved                                                                                                                                            
//             Licensed under the MIT License.
//                                                                           
//  Disclaimer:                                                                           
//    This project is provided without any guarantee and can be used for   
//    private and commercial purposes. Any use is at the user’s 
//    own risk and responsibility.
//
// -------------------------------------------------------------------------
TYPE ReadRobotDefaultDynamicsSendData EXTENDS CmdHeader: 
STRUCT
END_STRUCT
END_TYPE

{attribute 'pack_mode' := '1'} 
// ------------------------------------------------------------------------- 
//  SRCI Robot Library                                                
// ------------------------------------------------------------------------- 
//                                                                           
//  Object:      ReadRobotReferenceDynamicsOutCmd                                       
//  Author:      Thorsten Brach                                                
//  Date:        2024-08-09
//
//  Description:                                              
//   
//                                                                           
//  Copyright: 
//    (C) 2024 Thorsten Brach. All rights reserved                                                                                                                                            
//             Licensed under the MIT License.
//                                                                           
//  Disclaimer:                                                                           
//    This project is provided without any guarantee and can be used for   
//    private and commercial purposes. Any use is at the user’s 
//    own risk and responsibility.
//
// -------------------------------------------------------------------------
TYPE ReadRobotReferenceDynamicsOutCmd :
STRUCT
  /// Reference dynamics values according to Table 6-109.
  DynamicValues      : ReferenceDynamics;
END_STRUCT
END_TYPE

{attribute 'pack_mode' := '1'} 
// ------------------------------------------------------------------------- 
//  SRCI Robot Library                                                
// ------------------------------------------------------------------------- 
//                                                                           
//  Object:      ReadRobotReferenceDynamicsParCmd                                       
//  Author:      Thorsten Brach                                                
//  Date:        2024-08-09
//
//  Description:                                              
//   
//                                                                           
//  Copyright: 
//    (C) 2024 Thorsten Brach. All rights reserved                                                                                                                                            
//             Licensed under the MIT License.
//                                                                           
//  Disclaimer:                                                                           
//    This project is provided without any guarantee and can be used for   
//    private and commercial purposes. Any use is at the user’s 
//    own risk and responsibility.
//
// -------------------------------------------------------------------------
TYPE ReadRobotReferenceDynamicsParCmd :
STRUCT
END_STRUCT
END_TYPE

{attribute 'pack_mode' := '1'} 
// ------------------------------------------------------------------------- 
//  SRCI Robot Library                                                
// ------------------------------------------------------------------------- 
//                                                                           
//  Object:      ReadRobotReferenceDynamicsRecvData                                       
//  Author:      Thorsten Brach                                                
//  Date:        2024-08-09
//
//  Description:                                              
//   
//                                                                           
//  Copyright: 
//    (C) 2024 Thorsten Brach. All rights reserved                                                                                                                                            
//             Licensed under the MIT License.
//                                                                           
//  Disclaimer:                                                                           
//    This project is provided without any guarantee and can be used for   
//    private and commercial purposes. Any use is at the user’s 
//    own risk and responsibility.
//
// -------------------------------------------------------------------------
TYPE ReadRobotReferenceDynamicsRecvData EXTENDS RspHeader :
STRUCT
  /// Timestamp
  Timestamp             : IEC_TIMESTAMP;
  /// Path velocity [mm/s](tangent) at 100%
  /// • <0: (default) - Do not change values
  /// • ≥0: Change values according to input value
  VelocityReference     : REAL;
  /// Path acceleration [mm/s2] at 100%
  /// • <0: (default) - Do not change values
  /// • ≥0: Change values according to input value
  AccelerationReference : REAL;
  /// Path deceleration [mm/s2] at 100%
  /// • <0: (default) - Do not change values
  /// • ≥0: Change values according to input value
  DecelerationReference : REAL;
  /// Jerk [mm/s3] at 100%
  /// • <0: (default) - Do not change values
  /// • ≥0: Change values according to input value
  JerkReference        : REAL;  
  /// The status bit "DataChanged" represents the modification state 
  DataChanged          : BOOL;
END_STRUCT
END_TYPE

{attribute 'pack_mode' := '1'}
// ------------------------------------------------------------------------- 
//  SRCI Robot Library                                                
// ------------------------------------------------------------------------- 
//                                                                           
//  Object:      ReadRobotReferenceDynamicsSendData                                       
//  Author:      Thorsten Brach                                                
//  Date:        2024-08-09
//
//  Description:                                              
//   
//                                                                           
//  Copyright: 
//    (C) 2024 Thorsten Brach. All rights reserved                                                                                                                                            
//             Licensed under the MIT License.
//                                                                           
//  Disclaimer:                                                                           
//    This project is provided without any guarantee and can be used for   
//    private and commercial purposes. Any use is at the user’s 
//    own risk and responsibility.
//
// -------------------------------------------------------------------------
TYPE ReadRobotReferenceDynamicsSendData EXTENDS CmdHeader: 
STRUCT
END_STRUCT
END_TYPE

{attribute 'pack_mode' := '1'} 
// ------------------------------------------------------------------------- 
//  SRCI Robot Library                                                
// ------------------------------------------------------------------------- 
//                                                                           
//  Object:      ReadRobotSWLimitsOutCmd                                       
//  Author:      Thorsten Brach                                                
//  Date:        2024-08-09
//
//  Description:                                              
//   
//                                                                           
//  Copyright: 
//    (C) 2024 Thorsten Brach. All rights reserved                                                                                                                                            
//             Licensed under the MIT License.
//                                                                           
//  Disclaimer:                                                                           
//    This project is provided without any guarantee and can be used for   
//    private and commercial purposes. Any use is at the user’s 
//    own risk and responsibility.
//
// -------------------------------------------------------------------------
TYPE ReadRobotSWLimitsOutCmd :
STRUCT
  /// DLimits for joints and external axes according to Table 6-173.
  LimitValues        : SWLimits;
END_STRUCT
END_TYPE

{attribute 'pack_mode' := '1'} 
// ------------------------------------------------------------------------- 
//  SRCI Robot Library                                                
// ------------------------------------------------------------------------- 
//                                                                           
//  Object:      ReadRobotSWLimitsParCmd                                       
//  Author:      Thorsten Brach                                                
//  Date:        2024-08-09
//
//  Description:                                              
//   
//                                                                           
//  Copyright: 
//    (C) 2024 Thorsten Brach. All rights reserved                                                                                                                                            
//             Licensed under the MIT License.
//                                                                           
//  Disclaimer:                                                                           
//    This project is provided without any guarantee and can be used for   
//    private and commercial purposes. Any use is at the user’s 
//    own risk and responsibility.
//
// -------------------------------------------------------------------------
TYPE ReadRobotSWLimitsParCmd :
STRUCT
END_STRUCT
END_TYPE

{attribute 'pack_mode' := '1'} 
// ------------------------------------------------------------------------- 
//  SRCI Robot Library                                                
// ------------------------------------------------------------------------- 
//                                                                           
//  Object:      ReadRobotSWLimitsRecvData                                       
//  Author:      Thorsten Brach                                                
//  Date:        2024-08-09
//
//  Description:                                              
//   
//                                                                           
//  Copyright: 
//    (C) 2024 Thorsten Brach. All rights reserved                                                                                                                                            
//             Licensed under the MIT License.
//                                                                           
//  Disclaimer:                                                                           
//    This project is provided without any guarantee and can be used for   
//    private and commercial purposes. Any use is at the user’s 
//    own risk and responsibility.
//
// -------------------------------------------------------------------------
TYPE ReadRobotSWLimitsRecvData EXTENDS RspHeader :
STRUCT
  /// DLimits for joints and external axes according to Table 6-173.
  LimitValues        : SWLimits;
  /// The status bit "DataChanged" represents the modification state 
  DataChanged : BOOL;
END_STRUCT
END_TYPE

{attribute 'pack_mode' := '1'}
// ------------------------------------------------------------------------- 
//  SRCI Robot Library                                                
// ------------------------------------------------------------------------- 
//                                                                           
//  Object:      ReadRobotSWLimitsSendData                                       
//  Author:      Thorsten Brach                                                
//  Date:        2024-08-09
//
//  Description:                                              
//   
//                                                                           
//  Copyright: 
//    (C) 2024 Thorsten Brach. All rights reserved                                                                                                                                            
//             Licensed under the MIT License.
//                                                                           
//  Disclaimer:                                                                           
//    This project is provided without any guarantee and can be used for   
//    private and commercial purposes. Any use is at the user’s 
//    own risk and responsibility.
//
// -------------------------------------------------------------------------
TYPE ReadRobotSWLimitsSendData EXTENDS CmdHeader: 
STRUCT
END_STRUCT
END_TYPE

{attribute 'pack_mode' := '1'} 
// ------------------------------------------------------------------------- 
//  SRCI Robot Library                                                
// ------------------------------------------------------------------------- 
//                                                                           
//  Object:      ReadSystemVariableOutCmd                                       
//  Author:      Thorsten Brach                                                
//  Date:        2024-08-09
//
//  Description:                                              
//   
//                                                                           
//  Copyright: 
//    (C) 2024 Thorsten Brach. All rights reserved                                                                                                                                            
//             Licensed under the MIT License.
//                                                                           
//  Disclaimer:                                                                           
//    This project is provided without any guarantee and can be used for   
//    private and commercial purposes. Any use is at the user’s 
//    own risk and responsibility.
//
// -------------------------------------------------------------------------
TYPE ReadSystemVariableOutCmd :
STRUCT
  /// Unique system-generated ID of the "Action" when the function is triggered.
  /// • >0: The "Action" is started by the trigger function with identical FollowID.
  /// • <0: The "Action" is stopped by the trigger function with identical FollowID.
  /// For more information see chapter 5.5.12.4 EmitterID, ListenerID, FollowID and OriginID
  OriginID           : INT;
  /// Relates to ListenerID >0
  /// Number of successful trigger -based command invocations
  /// For more information refer to chapter 5.5.12.4.
  InvocationCounter  : USINT;
  
  /// Parameter data type as specified in Table 6-613.
  DataType           : ARRAY[0..7] OF USINT;
  /// Parameter data addressed by input values of ParameterID[0] and SubParameterID[0]
  Data_0             : ARRAY[0..3] OF BYTE;
  /// Parameter data addressed by input values of ParameterID[1] and SubParameterID[1]
  Data_1             : ARRAY[0..3] OF BYTE;
  /// Parameter data addressed by input values of ParameterID[2] and SubParameterID[2]
  Data_2             : ARRAY[0..3] OF BYTE;
  /// Parameter data addressed by input values of ParameterID[3] and SubParameterID[3]
  Data_3             : ARRAY[0..3] OF BYTE;
  /// Parameter data addressed by input values of ParameterID[4] and SubParameterID[4]
  Data_4             : ARRAY[0..3] OF BYTE;
  /// Parameter data addressed by input values of ParameterID[5] and SubParameterID[5]
  Data_5             : ARRAY[0..3] OF BYTE;
  /// Parameter data addressed by input values of ParameterID[6] and SubParameterID[6]
  Data_6             : ARRAY[0..3] OF BYTE;
  /// Parameter data addressed by input values of ParameterID[7] and SubParameterID[7]
  Data_7             : ARRAY[0..3] OF BYTE;
END_STRUCT
END_TYPE

